// SIMATIC S7-200 SMART project (STEP 7-Micro/WIN SMART), CPU SR40

ORGANIZATION_BLOCK MAIN:OB1
TITLE=程序注释
BEGIN
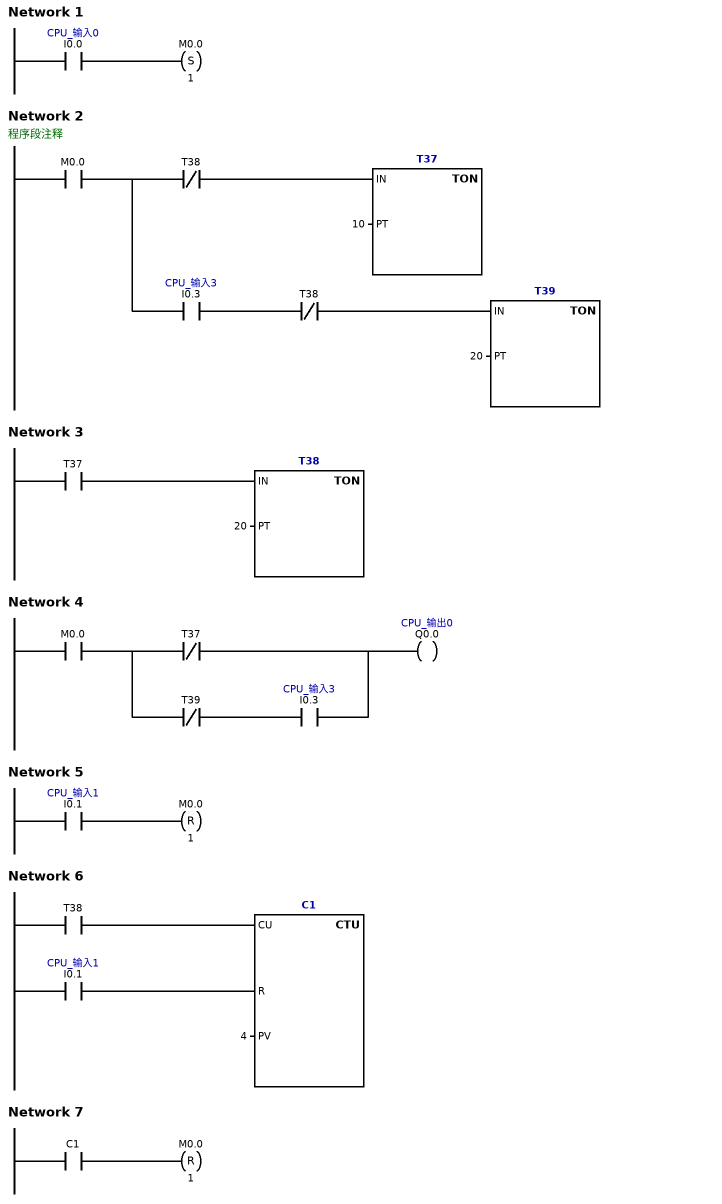
Network 1
LD     CPU_输入0:I0.0
S      M0.0, 1
Network 2
// 程序段注释
LD     M0.0
LPS
AN     T38
TON    T37, 10
LPP
A      CPU_输入3:I0.3
AN     T38
TON    T39, 20
Network 3
LD     T37
TON    T38, 20
Network 4
LD     M0.0
LDN    T37
LDN    T39
A      CPU_输入3:I0.3
OLD
ALD
=      CPU_输出0:Q0.0
Network 5
LD     CPU_输入1:I0.1
R      M0.0, 1
Network 6
LD     T38
LD     CPU_输入1:I0.1
CTU    C1, 4
Network 7
LD     C1
R      M0.0, 1
END_ORGANIZATION_BLOCK
